FUNCTION FC_5strConcat : T_DEFAULT_STR		// Concatenates 4 strings
VAR_INPUT
	iStr1:		T_DEFAULT_STR;
	iStr2:		T_DEFAULT_STR;
	iStr3:		T_DEFAULT_STR;
	iStr4:		T_DEFAULT_STR;
	iStr5:		T_DEFAULT_STR;
END_VAR

FC_5strConcat := CONCAT(FC_4strConcat(iStr1, iStr2, iStr3, iStr4),iStr5);

END_FUNCTION

(* stored: Version 1.1.0.1, ProductVersion 3.1.4026.18
   POU FC_5strConcat: Id {0acfa609-7eb4-476f-9646-e5afd72dd055}, SpecialFunc None *)
